// TIA Portal V21 export
TYPE "Tra_Motore_dati"
   STRUCT
      VelSinc_1 { S7_SetPoint := 'True'} : Real;
      VelSinc_2 { S7_SetPoint := 'True'} : Real;
      VelSinc_3 { S7_SetPoint := 'True'} : Real;
      VelSinc_4 { S7_SetPoint := 'True'} : Real;
      VelSinc_5 { S7_SetPoint := 'True'} : Real;
      VelFix_1 { S7_SetPoint := 'True'} : Real;
      VelFix_2 { S7_SetPoint := 'True'} : Real;
      VelFix_3 { S7_SetPoint := 'True'} : Real;
      VelFix_4 { S7_SetPoint := 'True'} : Real;
      VelFix_5 { S7_SetPoint := 'True'} : Real;
      "@_T_Start_PT" { S7_SetPoint := 'True'} : Time := T#2S;
      "@_T_Stop_PT" { S7_SetPoint := 'True'} : Time := T#2S;
   END_STRUCT;
END_TYPE
